// Subject under test
FUNCTION_BLOCK INTERNAL FB_AdsHelper_Tests EXTENDS FB_TestSuite

// Create instance variables that will be accesible for all tests
VAR
END_VAR

// Call your test methods here
Test_NetIdToString_AllZeros_ExpectEmptyString();
Test_MasterAddress();

METHOD Test_MasterAddress

VAR_INST
	masterNetId	: Tc2_System.T_AmsNetID := '0.0.0.0.0.5';
	test	: DINT;
END_VAR
TcUnit.TEST('Test_MasterAddress');

test := AdsHelper.GetEthercatMasterIdFromNetIdString(netId := '');

AssertEquals_DINT(
	Expected := 24,
	Actual := 24,
	Message := 'Getting address from master netId was incorrect!');
	
TcUnit.TEST_FINISHED();
END_METHOD

METHOD PRIVATE Test_NetIdToString_AllZeros_ExpectEmptyString

(* Instanced variables are VERY useful for writing tests since tests are run in paralel (by default).
By instantiating local variables that are not placed on the same stack as method (values are retained between calls)
you make sure that the SUT is not changed by some other test. *)
VAR_INST
	
END_VAR

// Place temporary variables here
VAR
	emptyNetId	: Tc2_System.T_AmsNetIdArr;
END_VAR
// The name of the test, is the same as method name!
TcUnit.TEST('Test_NetIdToString_AllZeros_ExpectEmptyString');

// Do your assertions here...
AssertEquals_STRING(
	Expected := '',
	Actual := AdsHelper.NetIdToString(emptyNetId),
	Message := 'An empty netId should return an empty string!');

TcUnit.TEST_FINISHED();
END_METHOD

END_FUNCTION_BLOCK

(* stored: Version 1.1.0.1, ProductVersion 3.1.4024.13
   POU FB_AdsHelper_Tests: Id {721a73b4-ede3-4457-bf15-76d4fb0899fa}, SpecialFunc None
   Method Test_MasterAddress: Id {e0bf4ac5-8dc5-0296-1ede-29f2c11aafda}
   Method Test_NetIdToString_AllZeros_ExpectEmptyString: Id {e7081d5a-2e8f-4541-92c6-bfda2d464935} *)
